PROGRAM OP120_Main
VAR
	OP120_Modeselection_FB: Mode_Selection_Block1;
	

	OP120_Vaccum1_Bit2: BOOL;
	OP120_Vaccum1_Bit6: BOOL;
	OP120_Vaccum1_Bit3: BOOL;
	OP120_Vaccum1_Bit4: BOOL;
	OP120_Vaccum1_Bit5: BOOL;
	OP120_Vaccum1_Bit7: BOOL;
	OP120_Vaccum_Byte2_bit0: BOOL;
	OP120_Vaccum_Byte2_bit1: BOOL;
	OP120_Vaccum_Byte2_bit2: BOOL;
	OP120_Vaccum_Byte2_bit3: BOOL;
	OP120_Vaccum_Byte2_bit4: BOOL;
	OP120_Vaccum_Byte2_bit5: BOOL;
	OP120_Vaccum_Byte2_bit6: BOOL;
	OP120_Vaccum_Byte2_bit7: BOOL;
	OP120_Vaccum2_Bit3: BOOL;
	OP120_Vaccum2_Bit4: BOOL;
	OP120_Vaccum2_Bit2: BOOL;
	OP120_Vaccum2_Bit5: BOOL;
	OP120_Vaccum2_Bit6: BOOL;
	OP120_Vaccum2_Bit7: BOOL;
	OP120_Vaccum2_Byte2_bit0: BOOL;
	OP120_Vaccum2_Byte2_bit1: BOOL;
	OP120_Vaccum2_Byte2_bit2: BOOL;
	OP120_Vaccum2_Byte2_bit3: BOOL;
	OP120_Vaccum2_Byte2_bit4: BOOL;
	OP120_Vaccum2_Byte2_bit5: BOOL;
	OP120_Vaccum2_Byte2_bit6: BOOL;
	OP120_Vaccum2_Byte2_bit7: BOOL;
END_VAR

op120_camera_FB();
OP120_Manual();
Op120_Error();

OP120_Initialization_Seq();
OP120_AutoSequence();
OP120_feed_Conveyor();
OP120_LockInsert_AutoSequence();

OP120_Sing_Auto_PRG();


IF (OP120_HMI_AutoMode AND NOT OP120_HMI_ManualMOde AND NOT OP120_HMI_StepMode) THEN
	OP120_Modeselection_FB.ModeWord:=1;
	ELSIF (NOT OP120_HMI_AutoMode AND OP120_HMI_ManualMOde AND NOT OP120_HMI_StepMode) THEN
		OP120_Modeselection_FB.ModeWord:=2;
	ELSIF  (NOT OP120_HMI_AutoMode AND NOT OP120_HMI_ManualMOde AND  OP120_HMI_StepMode) THEN
		OP120_Modeselection_FB.ModeWord:=3;
    ELSE   
		OP120_Modeselection_FB.ModeWord:=0;
END_IF
	





OP120_Modeselection_FB(
	ModeWord:= , 
	HomeConditionOK:=OP120_HomeCondition_OK , 
	OperationEnable:=OperationEnable , 
	StartPB:= , 
	SafetyAndNOError:=OperationEnable , 
	ModeAck:=TRUE , 
	HomingINProgress:= , 
	TempHomeOK:=OP120_Temp_Home_OK , 
	ResetPB:= , 
	AutoSelected=>OP120_AutoSelected , 
	ManualSelected=>OP120_ManualSelected , 
	StepSelected=>OP120_StepSelected , 
	ModeSelAck_Indication=> , 
	StatusDisplay=> , 
	AutoRunning:=OP120_AutoRunning , 
	StepRunning:=OP120_StepRunning , 
	StartEnable:=OP120_StartEnable , 
	MachineStop:=OP120_Machine_Stop );
	
	IF (OP120_AutoSelected OR  OP120_StepSelected ) THEN
		OP120_GVL.OP120_Auto:=TRUE;
		O120_ROB_MAN_AUTO_MODE_Q709_4:=TRUE;
		//OP120_SI_Dry_Run:=TRUE;
		OP120_Robo_Out6002:=1;
		
		ELSE
			OP120_GVL.OP120_Auto:=FALSE;
			O120_ROB_MAN_AUTO_MODE_Q709_4:=FALSE;
			OP120_Robo_Out6002:=0;
		END_IF
IF OP120_Auto AND NOT OP120_ManualSelected AND NOT OP120_HomeRunning THEN
	OP120_Robo_Out6001:=1;
END_IF
	
	(*OP120_Vaccum1_Bit0:=OP120_Vaccuum_IP_Port5_Byte1.7;
	OP120_Vaccum1_Bit1:=OP120_Vaccuum_IP_Port5_Byte1.6;
	OP120_Vaccum1_Bit2:=OP120_Vaccuum_IP_Port5_Byte1.5;
	OP120_Vaccum1_Bit3:=OP120_Vaccuum_IP_Port5_Byte1.4;
	OP120_Vaccum1_Bit4:=OP120_Vaccuum_IP_Port5_Byte1.3;
	OP120_Vaccum1_Bit5:=OP120_Vaccuum_IP_Port5_Byte1.2;
	OP120_Vaccum1_Bit6:=OP120_Vaccuum_IP_Port5_Byte1.1;
	OP120_Vaccum1_Bit7:=OP120_Vaccuum_IP_Port5_Byte1.0;
	
	OP120_Vaccum_Byte2_bit0:=OP120_Vaccuum_IP_Port5_Byte2.7;
	OP120_Vaccum_Byte2_bit1:=OP120_Vaccuum_IP_Port5_Byte2.6;
	OP120_Vaccum_Byte2_bit2:=OP120_Vaccuum_IP_Port5_Byte2.5;
	OP120_Vaccum_Byte2_bit3:=OP120_Vaccuum_IP_Port5_Byte2.4;
	OP120_Vaccum_Byte2_bit4:=OP120_Vaccuum_IP_Port5_Byte2.3;
	OP120_Vaccum_Byte2_bit5:=OP120_Vaccuum_IP_Port5_Byte2.2;
	OP120_Vaccum_Byte2_bit6:=OP120_Vaccuum_IP_Port5_Byte2.1;*)
	OP120_Vaccum1_Bit0:=OP120_Vaccuum_IP_Port5_Byte2.0;
	
(*OP120_Vaccum2_Bit0:=OP120_Vaccuum_IP_Port6_Byte1.7;
	OP120_Vaccum2_Bit1:=OP120_Vaccuum_IP_Port6_Byte1.6;
	OP120_Vaccum2_Bit2:=OP120_Vaccuum_IP_Port6_Byte1.5;
	OP120_Vaccum2_Bit3:=OP120_Vaccuum_IP_Port6_Byte1.4;
	OP120_Vaccum2_Bit4:=OP120_Vaccuum_IP_Port6_Byte1.3;
	OP120_Vaccum2_Bit5:=OP120_Vaccuum_IP_Port6_Byte1.2;
	OP120_Vaccum2_Bit6:=OP120_Vaccuum_IP_Port6_Byte1.1;
	OP120_Vaccum2_Bit7:=OP120_Vaccuum_IP_Port6_Byte1.0;
	
	OP120_Vaccum2_Byte2_bit0:=OP120_Vaccuum_IP_Port6_Byte2.7;
	OP120_Vaccum2_Byte2_bit1:=OP120_Vaccuum_IP_Port6_Byte2.6;
	OP120_Vaccum2_Byte2_bit2:=OP120_Vaccuum_IP_Port6_Byte2.5;
	OP120_Vaccum2_Byte2_bit3:=OP120_Vaccuum_IP_Port6_Byte2.4;
	OP120_Vaccum2_Byte2_bit4:=OP120_Vaccuum_IP_Port6_Byte2.3;
	OP120_Vaccum2_Byte2_bit5:=OP120_Vaccuum_IP_Port6_Byte2.2;
	OP120_Vaccum2_Byte2_bit6:=OP120_Vaccuum_IP_Port6_Byte2.1;*)
	OP120_Vaccum2_Bit0:=OP120_Vaccuum_IP_Port6_Byte2.0;

END_PROGRAM

(* stored: Version 1.1.0.1, ProductVersion 3.1.4024.11
   POU OP120_Main: Id {39e33e53-40d7-48b9-bca0-6c27b252bb43}, SpecialFunc None *)
